(* Logix 5000 project; controller Drives_Line1 1756-L72 rev 20.13; software revision 20.04; part 8 of 21 *)
(* tags used below, declared in another part *)
   IO_State_Pinch_1 : INT;
   IO_State_Tmp_Pinch_1 : INT;
   Pinchroll_1_RPMPerMPS : REAL;
   EntryCtrl : UDT_Control_Zone;
   In_Commands : UDT_Commands;
   In_Config : UDT_Config;
   LineCmd : UDT_Commands_Line;
   Out_Feedbacks : UDT_Fdbks;
   Out_Status : UDT_Status;
   Pinchroll_1 : UDT_Pinchroll;
   Pinchroll_2 : UDT_Pinchroll;
   TestConfig_Pinchroll_1 : UDT_Config_Pinch;
   Unwinder_1 : UDT_Unwinder;
   Unwinder_2 : UDT_Unwinder;
   zConfigFromMaster : BOOL;
   zPi : REAL;
   zSimulation : BOOL;
(* P12_Pinchroll_1, continued *)

ROUTINE R01_From_Master   (* ladder *)
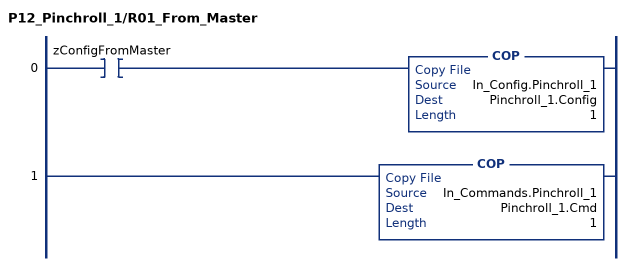
   0: XIC(zConfigFromMaster)COP(In_Config.Pinchroll_1,Pinchroll_1.Config,1);
   1: COP(In_Commands.Pinchroll_1,Pinchroll_1.Cmd,1);
END_ROUTINE

ROUTINE R02_From_Drive   (* ladder *)
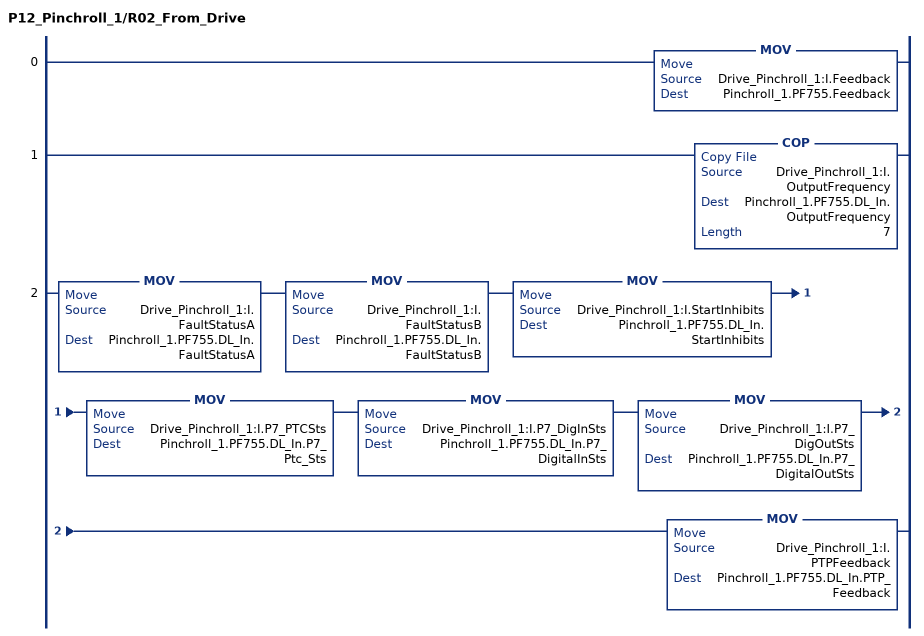
   0: MOV(Drive_Pinchroll_1:I.Feedback,Pinchroll_1.PF755.Feedback);
   1: COP(Drive_Pinchroll_1:I.OutputFrequency,Pinchroll_1.PF755.DL_In.OutputFrequency,7);
   2: MOV(Drive_Pinchroll_1:I.FaultStatusA,Pinchroll_1.PF755.DL_In.FaultStatusA)MOV(Drive_Pinchroll_1:I.FaultStatusB,Pinchroll_1.PF755.DL_In.FaultStatusB)MOV(Drive_Pinchroll_1:I.StartInhibits,Pinchroll_1.PF755.DL_In.StartInhibits)MOV(Drive_Pinchroll_1:I.P7_PTCSts,Pinchroll_1.PF755.DL_In.P7_Ptc_Sts)MOV(Drive_Pinchroll_1:I.P7_DigInSts,Pinchroll_1.PF755.DL_In.P7_DigitalInSts)MOV(Drive_Pinchroll_1:I.P7_DigOutSts,Pinchroll_1.PF755.DL_In.P7_DigitalOutSts)MOV(Drive_Pinchroll_1:I.PTPFeedback,Pinchroll_1.PF755.DL_In.PTP_Feedback);
END_ROUTINE

ROUTINE R03_Drive_Interface   (* ladder *)
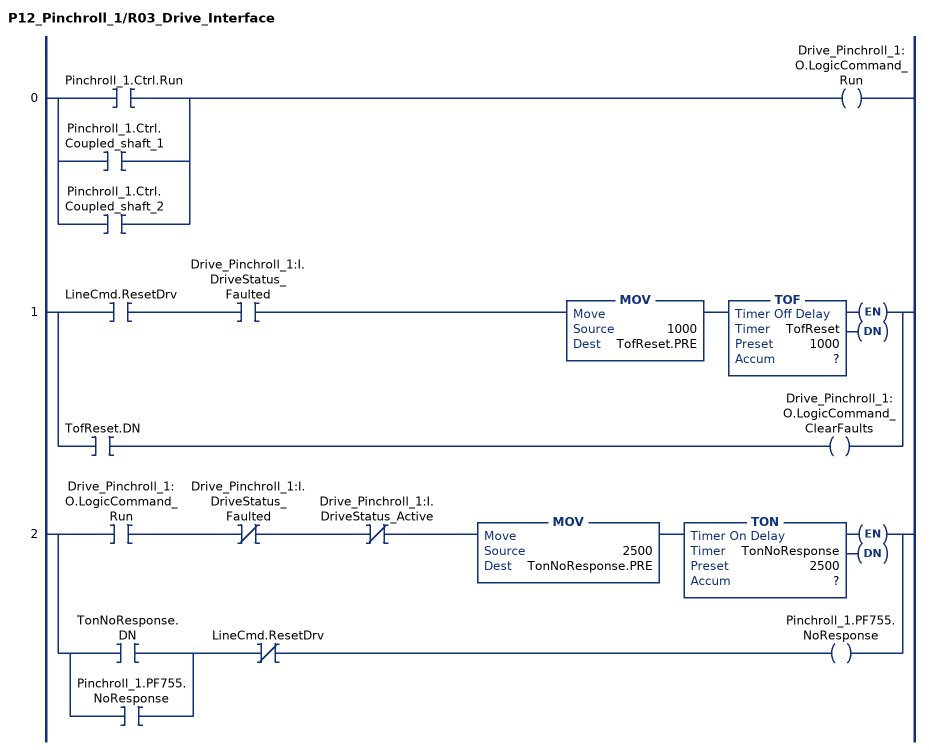
   0: [XIC(Pinchroll_1.Ctrl.Run) ,XIC(Pinchroll_1.Ctrl.Coupled_shaft_1) ,XIC(Pinchroll_1.Ctrl.Coupled_shaft_2) ]OTE(Drive_Pinchroll_1:O.LogicCommand_Run);
   1: [XIC(LineCmd.ResetDrv) XIC(Drive_Pinchroll_1:I.DriveStatus_Faulted) MOV(1000,TofReset.PRE) TOF(TofReset,?,?) ,XIC(TofReset.DN) OTE(Drive_Pinchroll_1:O.LogicCommand_ClearFaults) ];
   2: [XIC(Drive_Pinchroll_1:O.LogicCommand_Run) XIO(Drive_Pinchroll_1:I.DriveStatus_Faulted) XIO(Drive_Pinchroll_1:I.DriveStatus_Active) MOV(2500,TonNoResponse.PRE) TON(TonNoResponse,?,?) ,[XIC(TonNoResponse.DN) ,XIC(Pinchroll_1.PF755.NoResponse) ] XIO(LineCmd.ResetDrv) OTE(Pinchroll_1.PF755.NoResponse) ];
END_ROUTINE

ROUTINE R04_State   (* ladder *)
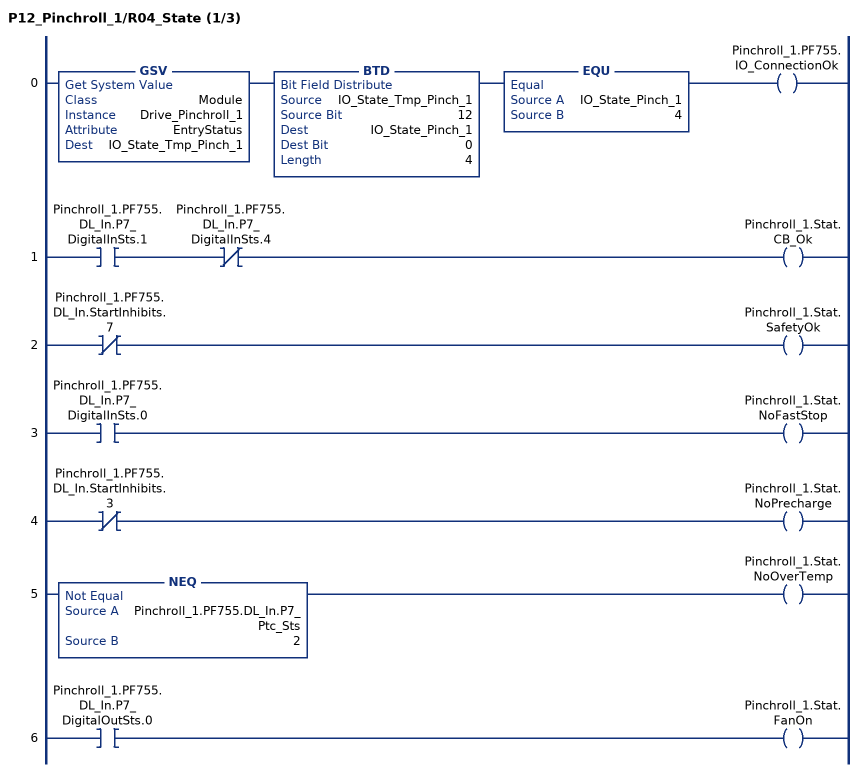
   0: GSV(Module,Drive_Pinchroll_1,EntryStatus,IO_State_Tmp_Pinch_1)BTD(IO_State_Tmp_Pinch_1,12,IO_State_Pinch_1,0,4)EQU(IO_State_Pinch_1,4)OTE(Pinchroll_1.PF755.IO_ConnectionOk);
   1: XIC(Pinchroll_1.PF755.DL_In.P7_DigitalInSts.1)XIO(Pinchroll_1.PF755.DL_In.P7_DigitalInSts.4)OTE(Pinchroll_1.Stat.CB_Ok);
   2: XIO(Pinchroll_1.PF755.DL_In.StartInhibits.7)OTE(Pinchroll_1.Stat.SafetyOk);
   3: XIC(Pinchroll_1.PF755.DL_In.P7_DigitalInSts.0)OTE(Pinchroll_1.Stat.NoFastStop);
   4: XIO(Pinchroll_1.PF755.DL_In.StartInhibits.3)OTE(Pinchroll_1.Stat.NoPrecharge);
   5: NEQ(Pinchroll_1.PF755.DL_In.P7_Ptc_Sts,2)OTE(Pinchroll_1.Stat.NoOverTemp);
   6: XIC(Pinchroll_1.PF755.DL_In.P7_DigitalOutSts.0)OTE(Pinchroll_1.Stat.FanOn);
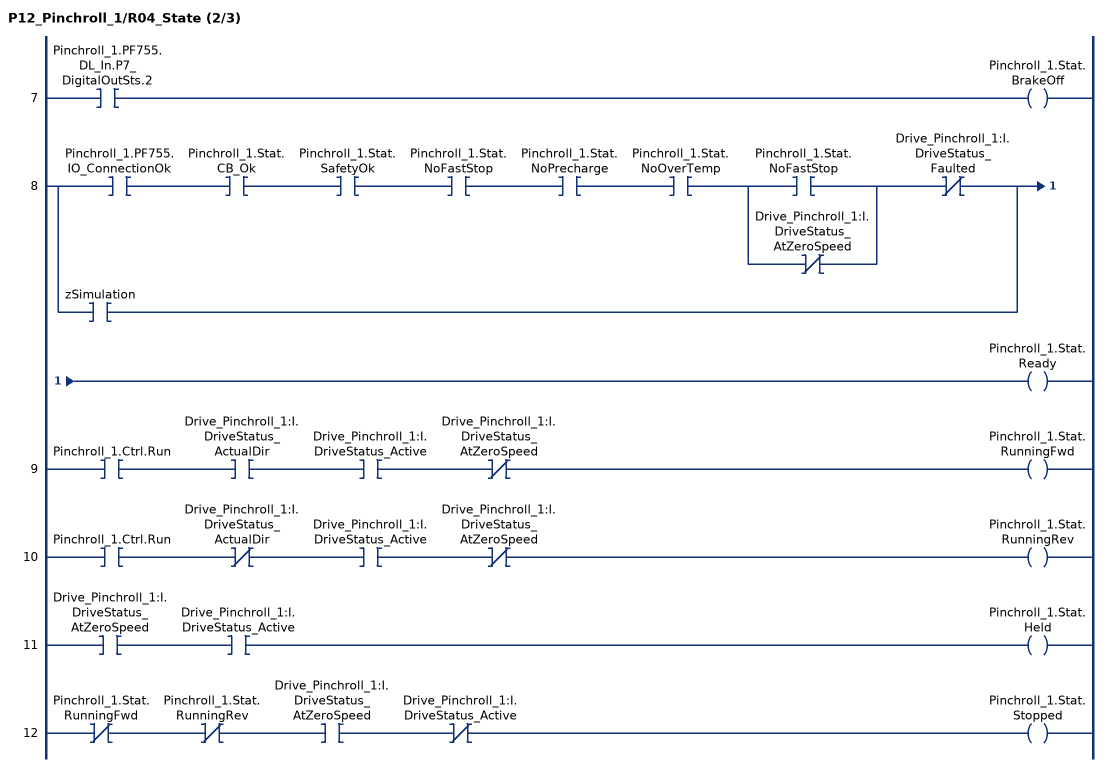
   7: XIC(Pinchroll_1.PF755.DL_In.P7_DigitalOutSts.2)OTE(Pinchroll_1.Stat.BrakeOff);
   8: [XIC(Pinchroll_1.PF755.IO_ConnectionOk) XIC(Pinchroll_1.Stat.CB_Ok) XIC(Pinchroll_1.Stat.SafetyOk) XIC(Pinchroll_1.Stat.NoFastStop) XIC(Pinchroll_1.Stat.NoPrecharge) XIC(Pinchroll_1.Stat.NoOverTemp) [XIC(Pinchroll_1.Stat.NoFastStop) ,XIO(Drive_Pinchroll_1:I.DriveStatus_AtZeroSpeed) ] XIO(Drive_Pinchroll_1:I.DriveStatus_Faulted) ,XIC(zSimulation) ]OTE(Pinchroll_1.Stat.Ready);
   9: XIC(Pinchroll_1.Ctrl.Run)XIC(Drive_Pinchroll_1:I.DriveStatus_ActualDir)XIC(Drive_Pinchroll_1:I.DriveStatus_Active)XIO(Drive_Pinchroll_1:I.DriveStatus_AtZeroSpeed)OTE(Pinchroll_1.Stat.RunningFwd);
   10: XIC(Pinchroll_1.Ctrl.Run)XIO(Drive_Pinchroll_1:I.DriveStatus_ActualDir)XIC(Drive_Pinchroll_1:I.DriveStatus_Active)XIO(Drive_Pinchroll_1:I.DriveStatus_AtZeroSpeed)OTE(Pinchroll_1.Stat.RunningRev);
   11: XIC(Drive_Pinchroll_1:I.DriveStatus_AtZeroSpeed)XIC(Drive_Pinchroll_1:I.DriveStatus_Active)OTE(Pinchroll_1.Stat.Held);
   12: XIO(Pinchroll_1.Stat.RunningFwd)XIO(Pinchroll_1.Stat.RunningRev)XIC(Drive_Pinchroll_1:I.DriveStatus_AtZeroSpeed)XIO(Drive_Pinchroll_1:I.DriveStatus_Active)OTE(Pinchroll_1.Stat.Stopped);
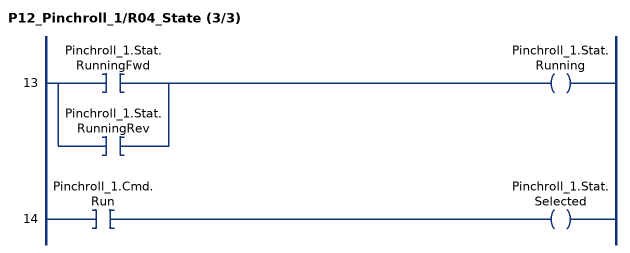
   13: [XIC(Pinchroll_1.Stat.RunningFwd) ,XIC(Pinchroll_1.Stat.RunningRev) ]OTE(Pinchroll_1.Stat.Running);
   14: XIC(Pinchroll_1.Cmd.Run)OTE(Pinchroll_1.Stat.Selected);
END_ROUTINE

ROUTINE R05_Control   (* ladder *)
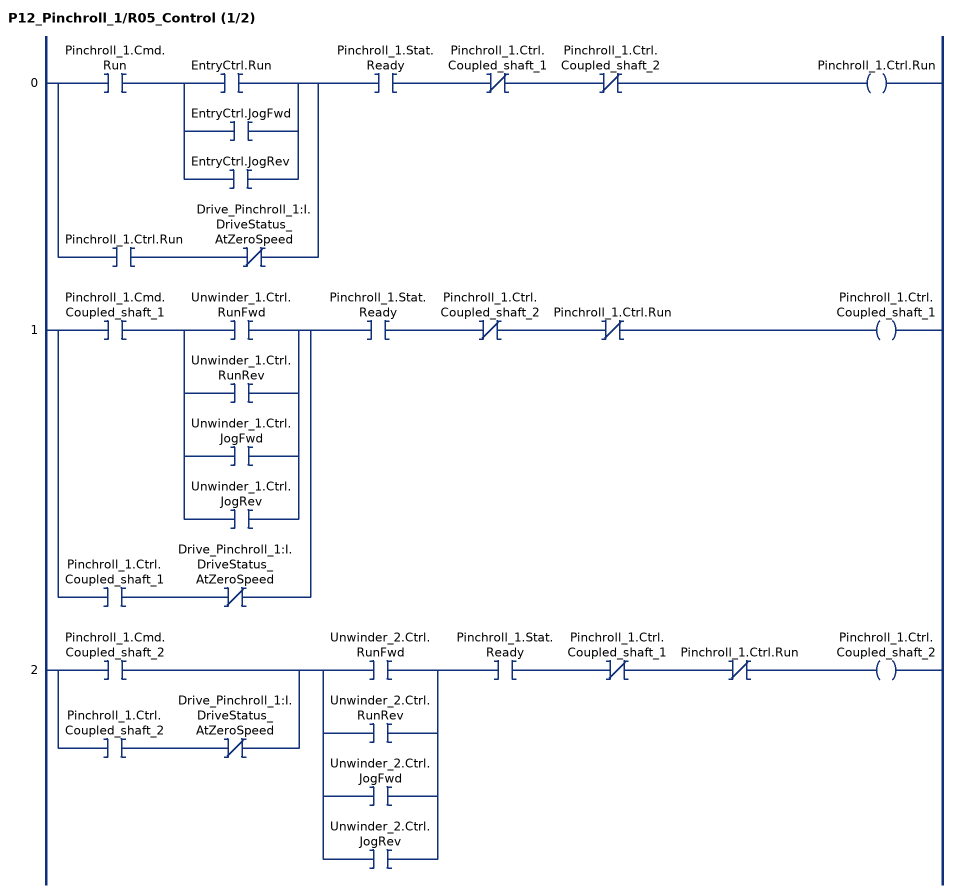
   0: [XIC(Pinchroll_1.Cmd.Run) [XIC(EntryCtrl.Run) ,XIC(EntryCtrl.JogFwd) ,XIC(EntryCtrl.JogRev) ] ,XIC(Pinchroll_1.Ctrl.Run) XIO(Drive_Pinchroll_1:I.DriveStatus_AtZeroSpeed) ]XIC(Pinchroll_1.Stat.Ready)XIO(Pinchroll_1.Ctrl.Coupled_shaft_1)XIO(Pinchroll_1.Ctrl.Coupled_shaft_2)OTE(Pinchroll_1.Ctrl.Run);
   1: [XIC(Pinchroll_1.Cmd.Coupled_shaft_1) [XIC(Unwinder_1.Ctrl.RunFwd) ,XIC(Unwinder_1.Ctrl.RunRev) ,XIC(Unwinder_1.Ctrl.JogFwd) ,XIC(Unwinder_1.Ctrl.JogRev) ] ,XIC(Pinchroll_1.Ctrl.Coupled_shaft_1) XIO(Drive_Pinchroll_1:I.DriveStatus_AtZeroSpeed) ]XIC(Pinchroll_1.Stat.Ready)XIO(Pinchroll_1.Ctrl.Coupled_shaft_2)XIO(Pinchroll_1.Ctrl.Run)OTE(Pinchroll_1.Ctrl.Coupled_shaft_1);
   2: [XIC(Pinchroll_1.Cmd.Coupled_shaft_2) ,XIC(Pinchroll_1.Ctrl.Coupled_shaft_2) XIO(Drive_Pinchroll_1:I.DriveStatus_AtZeroSpeed) ][XIC(Unwinder_2.Ctrl.RunFwd) ,XIC(Unwinder_2.Ctrl.RunRev) ,XIC(Unwinder_2.Ctrl.JogFwd) ,XIC(Unwinder_2.Ctrl.JogRev) ]XIC(Pinchroll_1.Stat.Ready)XIO(Pinchroll_1.Ctrl.Coupled_shaft_1)XIO(Pinchroll_1.Ctrl.Run)OTE(Pinchroll_1.Ctrl.Coupled_shaft_2);
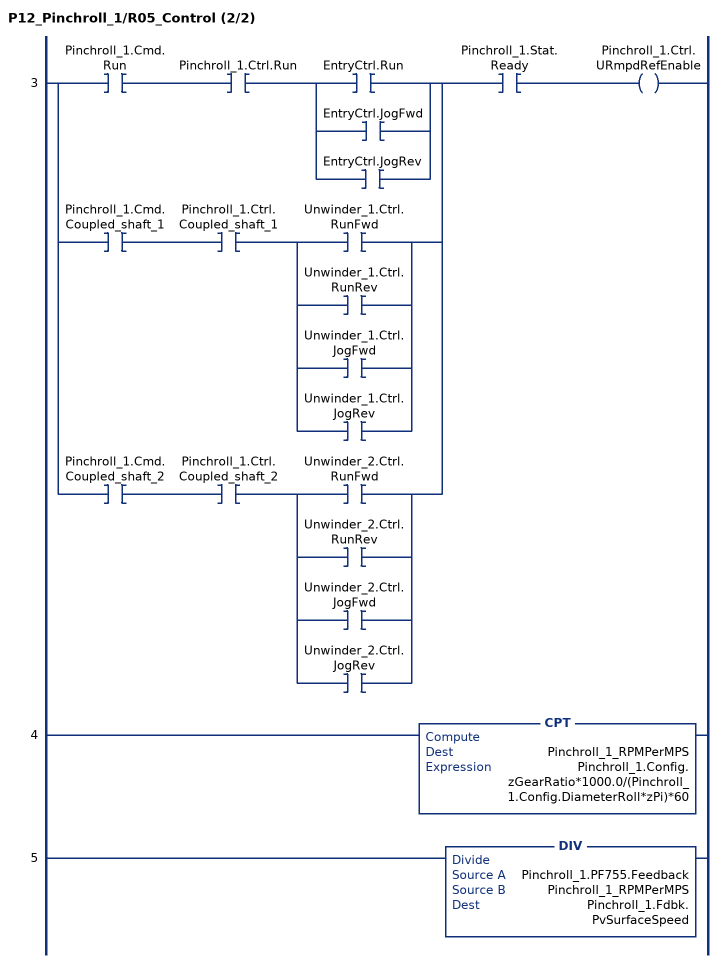
   3: [XIC(Pinchroll_1.Cmd.Run) XIC(Pinchroll_1.Ctrl.Run) [XIC(EntryCtrl.Run) ,XIC(EntryCtrl.JogFwd) ,XIC(EntryCtrl.JogRev) ] ,XIC(Pinchroll_1.Cmd.Coupled_shaft_1) XIC(Pinchroll_1.Ctrl.Coupled_shaft_1) [XIC(Unwinder_1.Ctrl.RunFwd) ,XIC(Unwinder_1.Ctrl.RunRev) ,XIC(Unwinder_1.Ctrl.JogFwd) ,XIC(Unwinder_1.Ctrl.JogRev) ] ,XIC(Pinchroll_1.Cmd.Coupled_shaft_2) XIC(Pinchroll_1.Ctrl.Coupled_shaft_2) [XIC(Unwinder_2.Ctrl.RunFwd) ,XIC(Unwinder_2.Ctrl.RunRev) ,XIC(Unwinder_2.Ctrl.JogFwd) ,XIC(Unwinder_2.Ctrl.JogRev) ] ]XIC(Pinchroll_1.Stat.Ready)OTE(Pinchroll_1.Ctrl.URmpdRefEnable);
   4: CPT(Pinchroll_1_RPMPerMPS,Pinchroll_1.Config.zGearRatio*1000.0/(Pinchroll_1.Config.DiameterRoll*zPi)*60);
   5: DIV(Pinchroll_1.PF755.Feedback,Pinchroll_1_RPMPerMPS,Pinchroll_1.Fdbk.PvSurfaceSpeed);
END_ROUTINE

ROUTINE R12_DriveRef   (* function block diagram *)
   SHEET 1   // Select speed reference
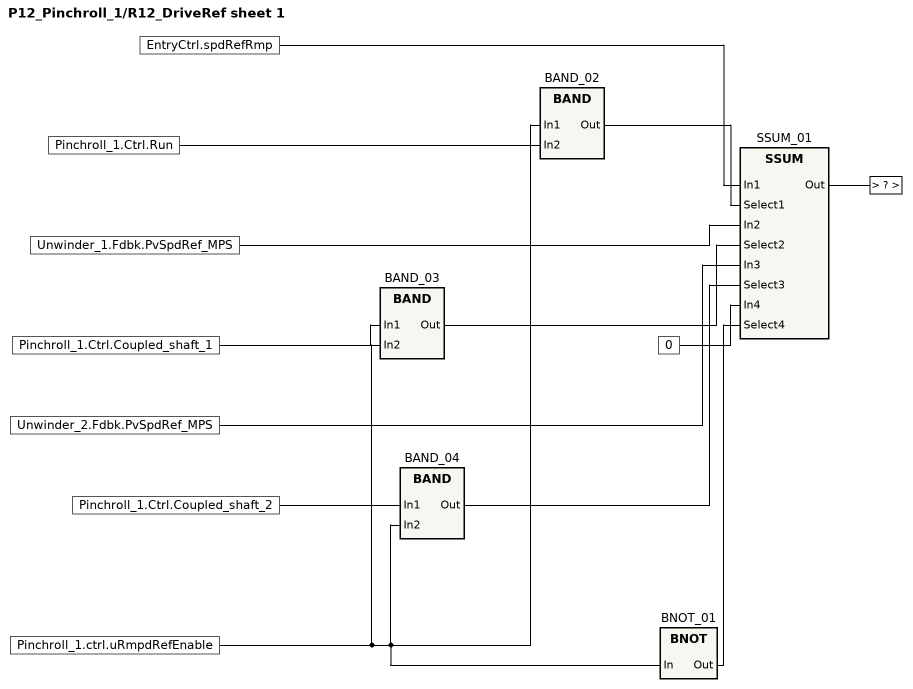
   BAND_03 : BAND(In1 := Pinchroll_1.Ctrl.Coupled_shaft_1, In2 := Pinchroll_1.ctrl.uRmpdRefEnable);
   BAND_04 : BAND(In1 := Pinchroll_1.Ctrl.Coupled_shaft_2, In2 := Pinchroll_1.ctrl.uRmpdRefEnable);
   BAND_02 : BAND(In1 := Pinchroll_1.ctrl.uRmpdRefEnable, In2 := Pinchroll_1.Ctrl.Run);
   BNOT_01 : BNOT(In := Pinchroll_1.ctrl.uRmpdRefEnable);
   SSUM_01 : SSUM(In1 := EntryCtrl.spdRefRmp, Select1 := BAND_02.Out, In2 := Unwinder_1.Fdbk.PvSpdRef_MPS, Select2 := BAND_03.Out, In3 := Unwinder_2.Fdbk.PvSpdRef_MPS, Select3 := BAND_04.Out, In4 := 0, Select4 := BNOT_01.Out);
   WIRE(?) := SSUM_01.Out;
   SHEET 2   // Final speed reference
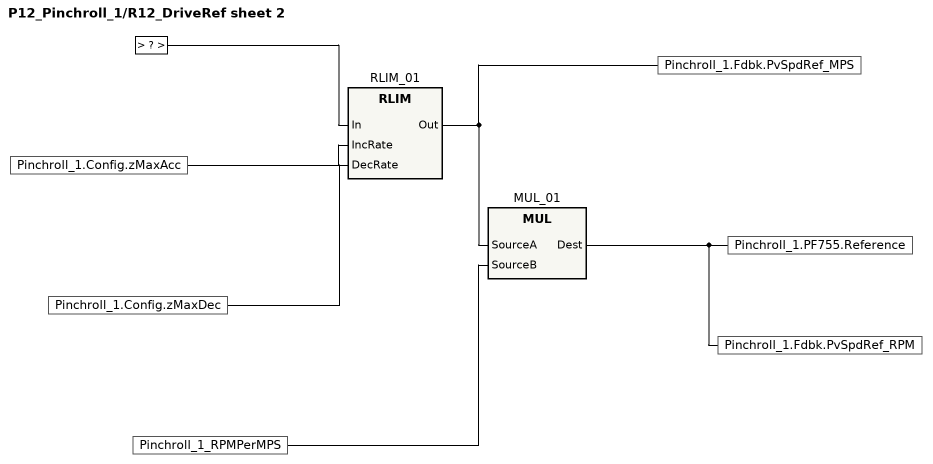
   RLIM_01 : RLIM(In := WIRE(?), IncRate := Pinchroll_1.Config.zMaxAcc, DecRate := Pinchroll_1.Config.zMaxDec);
   MUL_01 : MUL(SourceA := RLIM_01.Out, SourceB := Pinchroll_1_RPMPerMPS);
   Pinchroll_1.Fdbk.PvSpdRef_MPS := RLIM_01.Out;
   Pinchroll_1.Fdbk.PvSpdRef_RPM := MUL_01.Dest;
   Pinchroll_1.PF755.Reference := MUL_01.Dest;
   SHEET 3   // Speed reference synchronized
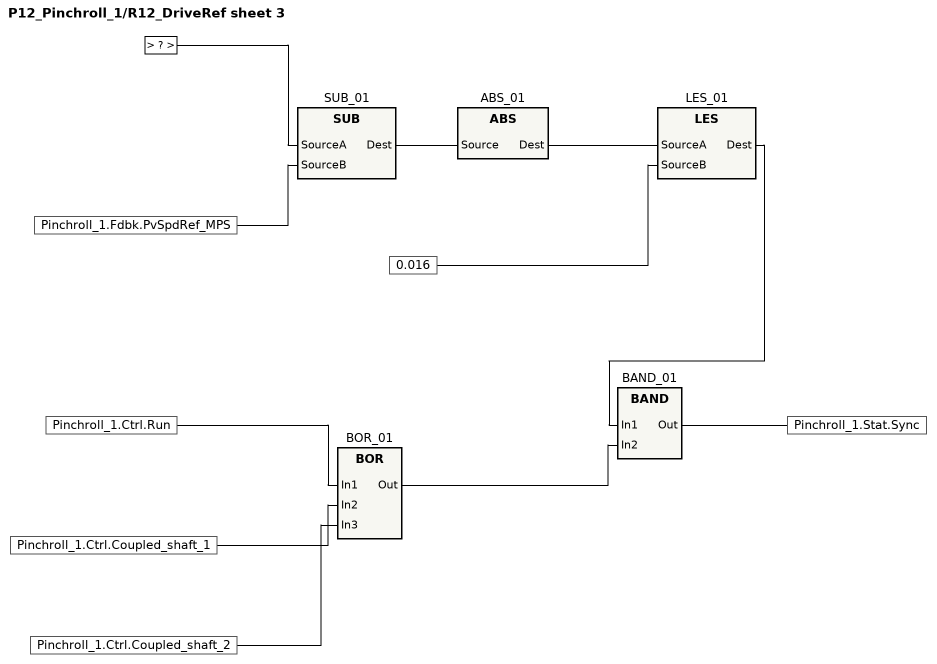
   SUB_01 : SUB(SourceA := WIRE(?), SourceB := Pinchroll_1.Fdbk.PvSpdRef_MPS);
   BOR_01 : BOR(In1 := Pinchroll_1.Ctrl.Run, In2 := Pinchroll_1.Ctrl.Coupled_shaft_1, In3 := Pinchroll_1.Ctrl.Coupled_shaft_2);
   ABS_01 : ABS(Source := SUB_01.Dest);
   LES_01 : LES(SourceA := ABS_01.Dest, SourceB := 0.016);
   BAND_01 : BAND(In1 := LES_01.Dest, In2 := BOR_01.Out);
   Pinchroll_1.Stat.Sync := BAND_01.Out;
END_ROUTINE

ROUTINE R98_ToDrive   (* ladder *)
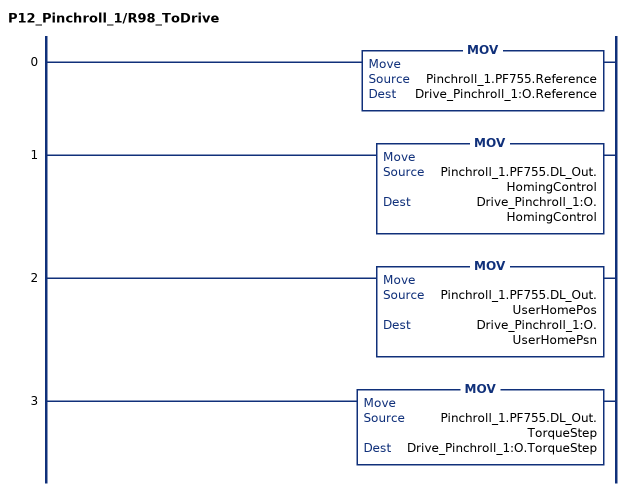
   0: MOV(Pinchroll_1.PF755.Reference,Drive_Pinchroll_1:O.Reference);
   1: MOV(Pinchroll_1.PF755.DL_Out.HomingControl,Drive_Pinchroll_1:O.HomingControl);
   2: MOV(Pinchroll_1.PF755.DL_Out.UserHomePos,Drive_Pinchroll_1:O.UserHomePsn);
   3: MOV(Pinchroll_1.PF755.DL_Out.TorqueStep,Drive_Pinchroll_1:O.TorqueStep);
END_ROUTINE

ROUTINE R999_Test   (* ladder *)
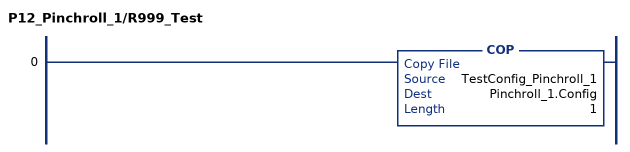
   0: COP(TestConfig_Pinchroll_1,Pinchroll_1.Config,1);
END_ROUTINE

ROUTINE R99_To_Master   (* ladder *)
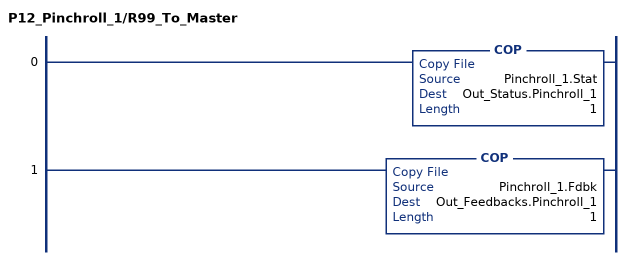
   0: COP(Pinchroll_1.Stat,Out_Status.Pinchroll_1,1);
   1: COP(Pinchroll_1.Fdbk,Out_Feedbacks.Pinchroll_1,1);
END_ROUTINE
END_PROGRAM

PROGRAM P13_Pinchroll_2   (* main routine R00_Main *)
VAR
   ABS_01 : FBD_MATH_ADVANCED;
   BAND_01 : FBD_BOOLEAN_AND := (In1 := 1, In3 := 1, In4 := 1, In5 := 1, In6 := 1, In7 := 1, In8 := 1);
   BAND_02 : FBD_BOOLEAN_AND := (In3 := 1, In4 := 1, In5 := 1, In6 := 1, In7 := 1, In8 := 1);
   BAND_03 : FBD_BOOLEAN_AND := (In3 := 1, In4 := 1, In5 := 1, In6 := 1, In7 := 1, In8 := 1);
   BAND_04 : FBD_BOOLEAN_AND := (In3 := 1, In4 := 1, In5 := 1, In6 := 1, In7 := 1, In8 := 1);
   BNOT_01 : FBD_BOOLEAN_NOT := (Out := 1);
   BOR_01 : FBD_BOOLEAN_OR;
   IO_State_Pinch_2 : INT := 4;
   IO_State_Tmp_Pinch_2 : INT := 16384;
   LES_01 : FBD_COMPARE := (SourceB := 0.016, Dest := 1);
   MUL_01 : FBD_MATH := (SourceB := 3181.732);
   Pinchroll_2_EncRes : DINT := 4096;
   Pinchroll_2_FB_Count_Old : DINT := 372815085;
   Pinchroll_2_Max_FB_Counts : DINT := 5120;
   Pinchroll_2_Rev_mm : REAL := 0.053028867;
   Pinchroll_2_RPMPerMPS : REAL := 3181.732;
   RLIM_01 : RATE_LIMITER := (IncRate := 0.1, DecRate := 0.1, RTSTime := 1, DeltaT := 0.05);
   SSUM_04 : SELECTED_SUMMER := (Gain1 := 1.0, Gain2 := 1.0, Gain3 := 1.0, Gain4 := 1.0, Select4 := 1, Gain5 := 1.0, Gain6 := 1.0, Gain7 := 1.0, Gain8 := 1.0);
   SUB_01 : FBD_MATH;
   TofReset : TIMER := (PRE := 1000, ACC := 1000);
   TonNoResponse : TIMER := (PRE := 2500);
   TonRefOn : TIMER := (PRE := 500);
   zPinchroll_2_Max_rev : REAL := 1500.0;
END_VAR

ROUTINE R00_Main   (* ladder *)
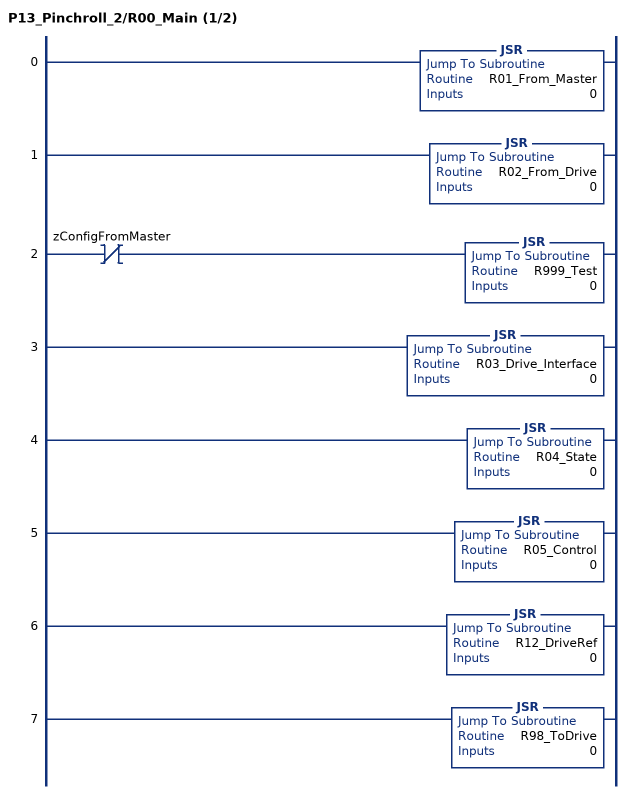
   0: JSR(R01_From_Master,0);
   1: JSR(R02_From_Drive,0);
   2: XIO(zConfigFromMaster)JSR(R999_Test,0);
   3: JSR(R03_Drive_Interface,0);
   4: JSR(R04_State,0);
   5: JSR(R05_Control,0);
   6: JSR(R12_DriveRef,0);
   7: JSR(R98_ToDrive,0);
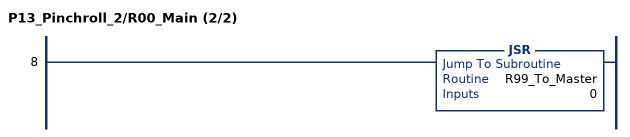
   8: JSR(R99_To_Master,0);
END_ROUTINE

ROUTINE R01_From_Master   (* ladder *)
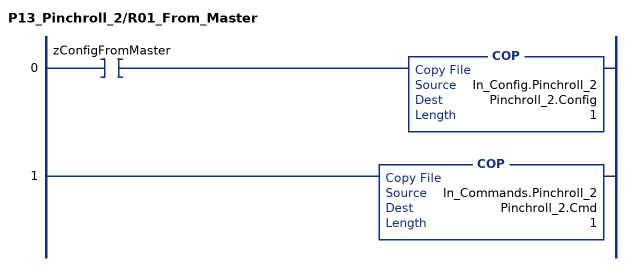
   0: XIC(zConfigFromMaster)COP(In_Config.Pinchroll_2,Pinchroll_2.Config,1);
   1: COP(In_Commands.Pinchroll_2,Pinchroll_2.Cmd,1);
END_ROUTINE

ROUTINE R02_From_Drive   (* ladder *)
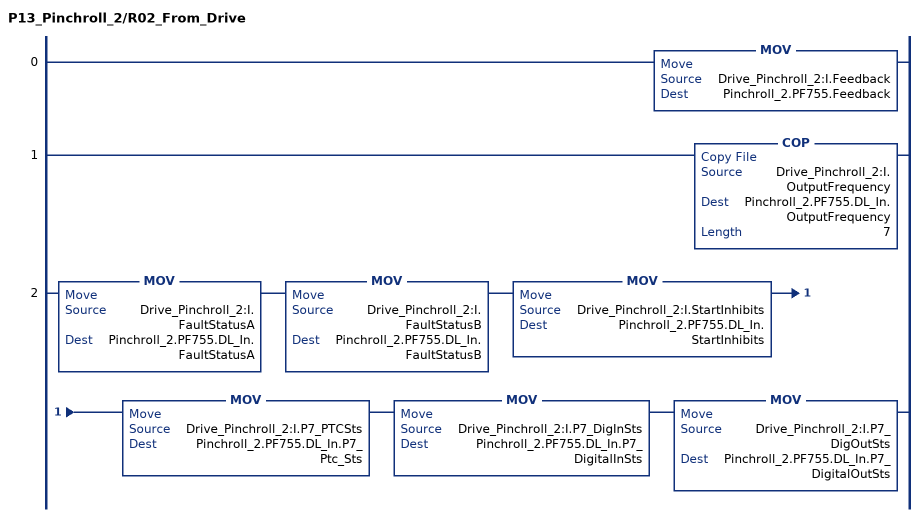
   0: MOV(Drive_Pinchroll_2:I.Feedback,Pinchroll_2.PF755.Feedback);
   1: COP(Drive_Pinchroll_2:I.OutputFrequency,Pinchroll_2.PF755.DL_In.OutputFrequency,7);
   2: MOV(Drive_Pinchroll_2:I.FaultStatusA,Pinchroll_2.PF755.DL_In.FaultStatusA)MOV(Drive_Pinchroll_2:I.FaultStatusB,Pinchroll_2.PF755.DL_In.FaultStatusB)MOV(Drive_Pinchroll_2:I.StartInhibits,Pinchroll_2.PF755.DL_In.StartInhibits)MOV(Drive_Pinchroll_2:I.P7_PTCSts,Pinchroll_2.PF755.DL_In.P7_Ptc_Sts)MOV(Drive_Pinchroll_2:I.P7_DigInSts,Pinchroll_2.PF755.DL_In.P7_DigitalInSts)MOV(Drive_Pinchroll_2:I.P7_DigOutSts,Pinchroll_2.PF755.DL_In.P7_DigitalOutSts);
END_ROUTINE
